(* CODESYS project retentivetimeroop_v0.0.1.1.library
   DefaultNamespace: RTimers
   Description: Standard library timers on TwinCAT count time by taking the difference between the current time from system timer and start time from system timer.
      While this is fine for most application, it is problematic for operations that require time to be retained even if the PLC is paused, stopped or turned off.
      For example, if a `TON` (Timer On-Delay) Timer is running and you stop the PLC Boot Project for a period of time, the `TON` will not resume from the point it was stopped.
      Instead it will skip time by the number of ms/secs/mins/hours it was stopped. 
      This makes it useless for applications such as tracking the length of time a PLC has been running or retaining persistent time.
      
      Retentive variants of the Standard library timers stop this from happen. They are based on PLC Task cycle time rather than system time. 
      This means they will simply stop counting when the PLC Task Cycle is stopped and will resume from where they left-off as soon as the task cycle picks up.
      All arguments behave in the same manner as those of the standard library.
   Author: Goodwill Mzumala & Victor Duran
   DocFormat: reStructuredText
   Title: Retentive Timers
   Version: 0.0.1.1
   Company: FisoThemes&Runtimevic
   Placeholder: Retentive Timers

Project tree, tasks and I/O mapping:
  libraries: Tc2_Standard, * (Beckhoff Automation GmbH); Tc2_System, * (Beckhoff Automation GmbH); Tc3_Module, * (Beckhoff Automation GmbH)
  DUTs/
    data type E_Timer_Type
    data type ST_Input
    data type ST_Output
    data type ST_PLC_TASK_INFORMATION
    data type ST_Setting
  Interfaces/
    interface I_Input: Pause, Start, StartTimer, StopTimer
    interface I_Output: Done, tElapsed
    interface I_Timer: Cyclic, Input, Output, Setting
  POUs/
    Function Block/
      Timers/
        function block FB_RStopwatch [ST]: Cyclic
        function block FB_RTimer [ST]: Cyclic
        function block FB_RTOF [ST]: Cyclic, Lerp
        function block FB_RTON [ST]: Cyclic, Lerp
        function block FB_RTP [ST]: Cyclic, Lerp
        function block FB_Stopwatch [ST]: Cyclic
        function block FB_Timer [ST]: Cyclic
      function block Timer [ST]: Cyclic, FB_exit, FB_init
      function block Timer_Abstract [ST]: Cyclic, Done, Input, Output, Pause, Setting, Start, StartTimer, StopTimer, tElapsed, tPreSet
    Functions/
      function F_Get_PLC_Task_Information [ST]
    program MAIN [ST]
  Project Information/
    function F_GetCompany [ST]
    function F_GetTitle [ST]
    function F_GetVersion [ST]
  Version/
    global variables Global_Version
*)

// DUTs/E_Timer_Type
{attribute 'qualified_only'}
{attribute 'strict'}
TYPE E_Timer_Type :
(
	RStopwatch := 0,
	RTimer,
	RTOF,
	RTON,
	RTP,
	Stopwatch,
	Timer,
	TOF,
	TON,
	TP
	
);
END_TYPE

// DUTs/ST_Input
TYPE ST_Input :
STRUCT
	bStart 		: BOOL;  // Starts timer with rising edge, resets timer with falling edge.
	bPause 		:  BOOL; // Pause Timer (TRUE), Only Pauses if IN := TRUE.
END_STRUCT
END_TYPE

// DUTs/ST_Output
TYPE ST_Output :
STRUCT
	bDone 		: BOOL; // Is TRUE, PT seconds after IN had a rising edge
	tElapsed 	: TIME; // Elapsed time
END_STRUCT
END_TYPE

// DUTs/ST_PLC_TASK_INFORMATION
TYPE ST_PLC_TASK_INFORMATION EXTENDS PlcTaskSystemInfo :
STRUCT
	tCycleTime 	: TIME; 	// Current task cycle time
	tlCycleTime : LTIME; 	// Current task cycle time in LTIME
END_STRUCT
END_TYPE

// DUTs/ST_Setting
TYPE ST_Setting :
STRUCT
	tPreSet 	: TIME; // Time to pass, before Q is set
END_STRUCT
END_TYPE

// Version/Global_Version
{attribute 'TcGenerated'}
{attribute 'no-analysis'}
{attribute 'linkalways'}
// This function has been automatically generated from the project information.
VAR_GLOBAL CONSTANT
	{attribute 'const_non_replaced'}
	stLibVersion_Retentive_Timers : ST_LibVersion := (iMajor := 0, iMinor := 0, iBuild := 1, iRevision := 1, nFlags := 0, sVersion := '0.0.1.1');
END_VAR

// Interfaces/I_Input
INTERFACE I_Input

METHOD Pause : I_Output
VAR_INPUT
	bPause 		:  BOOL; // Pause Timer (TRUE), Only Pauses if IN := TRUE.
END_VAR
END_METHOD

METHOD Start : I_Output
VAR_INPUT
	bStart 		: BOOL;  // Starts timer with rising edge, resets timer with falling edge.
END_VAR
END_METHOD

METHOD StartTimer : I_Output
VAR_INPUT
END_VAR
END_METHOD

METHOD StopTimer : I_Output
VAR_INPUT
END_VAR
END_METHOD

END_INTERFACE

// Interfaces/I_Output
INTERFACE I_Output

PROPERTY Done : BOOL
GET
END_GET
END_PROPERTY

PROPERTY tElapsed : TIME
GET
END_GET
END_PROPERTY

END_INTERFACE

// POUs/Function Block/Timer
{attribute 'hide_all_locals'}
FUNCTION_BLOCK Timer EXTENDS Timer_Abstract
VAR
	_eTimer         : E_Timer_Type;
	i_Timer			: I_Timer := 0;;
	
//	FB_RStopwatch 	: FB_RStopwatch;
//	FB_RTimer       : FB_RTimer;
//	FB_RTOF 		: FB_RTOF;
//	FB_RTON         : FB_RTON;
//	FB_RTP          : FB_RTP;
//	FB_Stopwatch 	: FB_Stopwatch;
//	FB_Timer        : FB_Timer;
	
	pRStopwatch 	: POINTER TO FB_RStopwatch;
	pRTimer       	: POINTER TO FB_RTimer;
	pRTOF 			: POINTER TO FB_RTOF;
	pRTON         	: POINTER TO FB_RTON;
	pRTP          	: POINTER TO FB_RTP;
	pStopwatch 		: POINTER TO FB_Stopwatch;
	pTimer        	: POINTER TO FB_Timer;
END_VAR

Cyclic();


METHOD Cyclic

//CASE _eTimer OF
	
//	E_Timer_Type.RStopwatch:
//		i_Timer   := FB_RStopwatch;
////	    pRStopwatch:= __NEW(FB_RStopwatch);
////		i_Timer   := pRStopwatch^;
		
////		//Release the memory
////		IF (pRStopwatch <> 0) THEN
////			__DELETE(pRStopwatch);
////			pRStopwatch := 0;
////		END_IF

//	E_Timer_Type.RTimer:
//		i_Timer   := FB_RTimer;

//	E_Timer_Type.RTOF:
//		i_Timer   := FB_RTOF;

//	E_Timer_Type.RTON:
//		i_Timer   := FB_RTON;

//	E_Timer_Type.RTP:
//		i_Timer   := FB_RTP;

//	E_Timer_Type.Stopwatch:
//		i_Timer   := FB_Stopwatch;

//	E_Timer_Type.Timer:
//		i_Timer   := FB_Timer;		
//END_CASE

IF i_Timer <> 0 THEN
	i_Timer.Input   REF= SUPER^._Input;
	i_Timer.Setting REF= SUPER^._Setting;
	i_Timer.Cyclic();
	SUPER^._Output := i_Timer.Output;
END_IF
END_METHOD

METHOD FB_exit : BOOL
VAR_INPUT
	bInCopyCode : BOOL; // if TRUE, the exit method is called for exiting an instance that is copied afterwards (online change).
END_VAR
IF (pRStopwatch <> 0) THEN
	__DELETE(pRStopwatch);
	pRStopwatch := 0;
END_IF

IF (pRTimer <> 0) THEN
	__DELETE(pRTimer);
	pRTimer := 0;
END_IF

IF (pRTOF <> 0) THEN
	__DELETE(pRTOF);
	pRTOF := 0;
END_IF

IF (pRTON <> 0) THEN
	__DELETE(pRTON);
	pRTON := 0;
END_IF

IF (pRTP <> 0) THEN
	__DELETE(pRTP);
	pRTP := 0;
END_IF

IF (pStopwatch <> 0) THEN
	__DELETE(pStopwatch);
	pStopwatch := 0;
END_IF

IF (pTimer <> 0) THEN
	__DELETE(pTimer);
	pTimer := 0;
END_IF
END_METHOD

METHOD FB_init : BOOL
VAR_INPUT
	bInitRetains : BOOL; // if TRUE, the retain variables are initialized (warm start / cold start)
	bInCopyCode : BOOL;  // if TRUE, the instance afterwards gets moved into the copy code (online change)
	eTimer      : E_Timer_Type;
END_VAR
THIS^._eTimer := eTimer;

CASE _eTimer OF
	
	E_Timer_Type.RStopwatch:
//		i_Timer   := FB_RStopwatch;
		pRStopwatch := __NEW(FB_RStopwatch);
		i_Timer := pRStopwatch^;

	E_Timer_Type.RTimer:
//		i_Timer   := FB_RTimer;
		pRTimer := __NEW(FB_RTimer);
		i_Timer := pRTimer^;

	E_Timer_Type.RTOF:
//		i_Timer   := FB_RTOF;
		pRTOF := __NEW(FB_RTOF);
		i_Timer := pRTOF^;

	E_Timer_Type.RTON:
//		i_Timer   := FB_RTON;
		pRTON := __NEW(FB_RTON);
		i_Timer := pRTON^;

	E_Timer_Type.RTP:
//		i_Timer   := FB_RTP;
		pRTP := __NEW(FB_RTP);
		i_Timer := pRTP^;

	E_Timer_Type.Stopwatch:
//		i_Timer   := FB_Stopwatch;
		pStopwatch := __NEW(FB_Stopwatch);
		i_Timer := pStopwatch^;

	E_Timer_Type.Timer:
//		i_Timer   := FB_Timer;
		pTimer := __NEW(FB_Timer);
		i_Timer := pTimer^;	
END_CASE
END_METHOD

END_FUNCTION_BLOCK

// POUs/Function Block/Timer_Abstract
{attribute 'enable_dynamic_creation'}
FUNCTION_BLOCK ABSTRACT Timer_Abstract IMPLEMENTS I_Timer, I_Input, I_Output
VAR_INPUT
END_VAR
VAR_OUTPUT
END_VAR
VAR
	_Setting 	: ST_Setting;
	_Input 		: ST_Input;
	_Output     : ST_Output;
END_VAR


METHOD ABSTRACT Cyclic
END_METHOD

PROPERTY Done : BOOL
GET
Done := _Output.bDone ;
END_GET
END_PROPERTY


PROPERTY Input : REFERENCE TO ST_Input
GET
Input REF= THIS^._Input ;
END_GET
SET
THIS^._Input := Input;
END_SET
END_PROPERTY


PROPERTY Output : REFERENCE TO ST_Output
GET
Output REF= THIS^._Output;
END_GET
END_PROPERTY

METHOD Pause : I_Output
VAR_INPUT
	bPause 		:  BOOL; // Pause Timer (TRUE), Only Pauses if IN := TRUE.
END_VAR
_Input.bPause := bPause;

Pause := THIS^;
END_METHOD


PROPERTY Setting : REFERENCE TO ST_Setting
GET
Setting REF= THIS^._Setting ;
END_GET
SET
THIS^._Setting := Setting;
END_SET
END_PROPERTY

METHOD Start : I_Output
VAR_INPUT
	bStart 		: BOOL;  // Starts timer with rising edge, resets timer with falling edge.
END_VAR
_Input.bStart := bStart;

Start := THIS^;
END_METHOD

METHOD StartTimer : I_Output
VAR_INPUT
END_VAR
_Input.bStart := TRUE;

StartTimer := THIS^;
END_METHOD

METHOD StopTimer : I_Output
VAR_INPUT
END_VAR
_Input.bStart := FALSE;

StopTimer := THIS^;
END_METHOD

PROPERTY tElapsed : TIME
GET
tElapsed := _Output.tElapsed; // Elapsed time
END_GET
END_PROPERTY

METHOD tPreSet
VAR_INPUT
	tPreSet 	: TIME; // Time to pass, before Q is set	
END_VAR
_Setting.tPreSet := tPreSet;
END_METHOD

END_FUNCTION_BLOCK

// Interfaces/I_Timer
INTERFACE I_Timer

METHOD Cyclic
END_METHOD

PROPERTY Input : REFERENCE TO ST_Input
GET
END_GET
SET
END_SET
END_PROPERTY

PROPERTY Output : REFERENCE TO ST_Output
GET
END_GET
END_PROPERTY

PROPERTY Setting : REFERENCE TO ST_Setting
GET
END_GET
SET
END_SET
END_PROPERTY

END_INTERFACE

// POUs/Function Block/Timers/FB_RStopwatch
// Retentive stopwatch
{attribute 'enable_dynamic_creation'}
FUNCTION_BLOCK INTERNAL FB_RStopwatch EXTENDS Timer_Abstract
//VAR_INPUT
//	bStart 			: BOOL;
//END_VAR
//VAR_OUTPUT
//	tElapsed 		: TIME;
//END_VAR
VAR
	stPLC_Task_Info : ST_PLC_TASK_INFORMATION;
	tAccumulator 	: TIME;
	fbTON 			: FB_RTON;
END_VAR


METHOD Cyclic
IF SUPER^._Input.bStart THEN stPLC_Task_Info := F_Get_PLC_Task_Information(); END_IF

//fbTON(tPreSet := stPLC_Task_Info.tCycleTime*2 + tAccumulator);
//fbTON(bStart := SUPER^._Input.bStart AND NOT(fbTON.output.bDone));
fbTON._Setting.tPreSet := stPLC_Task_Info.tCycleTime*2 + tAccumulator;
fbTON._Input.bStart := SUPER^._Input.bStart AND NOT(fbTON.output.bDone);
fbTON.Cyclic();

tAccumulator := fbTON.Output.tElapsed; 

IF SUPER^._Input.bStart THEN Output.tElapsed := tAccumulator; END_IF
END_METHOD

END_FUNCTION_BLOCK

// POUs/Function Block/Timers/FB_RTON
(* Retentive Timer On-Delay - implements a timer-on delay that persists if PLC cycle is stopped. 
When the input gets TRUE, elapsed time ET will run until also the output Q becomes TRUE. 
*)
{attribute 'enable_dynamic_creation'}
FUNCTION_BLOCK INTERNAL FB_RTON EXTENDS Timer_Abstract
//VAR_INPUT
//	bStart 				: BOOL; // Starts timer with rising edge, resets timer with falling edge
//	tPreSet 			: TIME; // Time to pass, before Q is set
//END_VAR
//VAR_OUTPUT
//	bDone 				: BOOL; // Is TRUE, PT seconds after IN had a rising edge
//	tElapsed 			: TIME; // Elapsed time
//END_VAR
VAR
	stPLC_Task_Info 	: ST_PLC_TASK_INFORMATION;
	tAccumulator 		: TIME;
	nLast_Cycle_Count 	: UDINT;
END_VAR


METHOD Cyclic
IF SUPER^._Input.bStart THEN
	stPLC_Task_Info := F_Get_PLC_Task_Information();
	SUPER^._Output.bDone := SUPER^._Output.tElapsed >= SUPER^._Setting.tPreSet;
	
	IF NOT(SUPER^._Output.bDone) AND ((nLast_Cycle_Count <> stPLC_Task_Info.CycleCount) OR nLast_Cycle_Count = 0) THEN
		tAccumulator := tAccumulator + stPLC_Task_Info.tCycleTime; 
		SUPER^._Output.tElapsed := LIMIT(T#0MS, THIS^.Lerp(T#0MS, SUPER^._Setting.tPreSet, TO_REAL(tAccumulator)/TO_REAL(SUPER^._Setting.tPreSet))-stPLC_Task_Info.tCycleTime, SUPER^._Setting.tPreSet);
		nLast_Cycle_Count := stPLC_Task_Info.CycleCount;
		END_IF
	RETURN;
	END_IF
tAccumulator := SUPER^._Output.tElapsed := T#0MS; SUPER^._Output.bDone := FALSE;
END_METHOD

// Linear interpolation (Lerp) - this method interpolates values between 2 time points.
METHOD PRIVATE Lerp : TIME
VAR_INPUT
	tStart 	: TIME := T#0MS; 
	tFinish : TIME;
	fPercentage : REAL; // Value must be between 0 and 1
END_VAR
// Lerp(Start, Finish, Percentage) = Start + (Finish - Start)*Percentage
Lerp := TO_TIME(TO_REAL(tStart) + TO_REAL(tFinish - tStart)*fPercentage);
END_METHOD

END_FUNCTION_BLOCK

// POUs/Functions/F_Get_PLC_Task_Information
(* Gets the infomation of the task the function is currently called on.
.. _More: https://infosys.beckhoff.com/english.php?content=../content/1033/globaldatatypes/714818699.html&id=
*)
FUNCTION F_Get_PLC_Task_Information : ST_PLC_TASK_INFORMATION
VAR_INPUT
END_VAR
VAR
	fbCurrent_Task_Index  	: GETCURTASKINDEX;
	st_TaskInfo 			: PlcTaskSystemInfo;
	stTask_Info 			: ST_PLC_TASK_INFORMATION;
END_VAR

fbCurrent_Task_Index();
st_TaskInfo 						:= TwinCAT_SystemInfoVarList._TaskInfo[fbCurrent_Task_Index.index];

stTask_Info.AdsPort 				:= st_TaskInfo.AdsPort;
stTask_Info.CycleCount 				:= st_TaskInfo.CycleCount;
stTask_Info.CycleTime 				:= st_TaskInfo.CycleTime;
stTask_Info.CycleTimeExceeded 		:= st_TaskInfo.CycleTimeExceeded;
stTask_Info.DcTaskTime 				:= st_TaskInfo.DcTaskTime;
stTask_Info.FirstCycle				:= st_TaskInfo.FirstCycle;
stTask_Info.InCallAfterOutputUpdate := st_TaskInfo.InCallAfterOutputUpdate;
stTask_Info.LastExecTime 			:= st_TaskInfo.LastExecTime;
stTask_Info.ObjId 					:= st_TaskInfo.ObjId;
stTask_Info.Priority 				:= st_TaskInfo.Priority;
stTask_Info.RTViolation 			:= st_TaskInfo.RTViolation;
stTask_Info.TaskName 				:= st_TaskInfo.TaskName;
stTask_Info.tlCycleTime 			:= TO_LTIME(st_TaskInfo.CycleTime*100);
stTask_Info.tCycleTime 				:= TO_TIME(stTask_Info.tlCycleTime);

F_Get_PLC_Task_Information 		:= stTask_Info;

END_FUNCTION

// POUs/Function Block/Timers/FB_RTimer
// Retentive Pausable Timer Function Block
{attribute 'enable_dynamic_creation'}
FUNCTION_BLOCK INTERNAL FB_RTimer EXTENDS Timer_Abstract
//VAR_INPUT
//    bStart 			: BOOL; // Start (TRUE) or Stop (FALSE) Timer 
//	bPause 			: BOOL; // Pause Timer (TRUE), Only Pauses if IN := TRUE
//    tPreSet			: TIME; // Set Time
//END_VAR
//VAR_OUTPUT
//    bDone 			: BOOL;	// Becomes TRUE after Set Time has passed
//    tElapsed 		: TIME; // Time Elapsed
//END_VAR
VAR
	fbRTON 			: FB_RTON;
END_VAR


METHOD Cyclic
IF NOT(SUPER^._Input.bStart) THEN 
	//fbRTON(bStart := FALSE, bDone => SUPER^._Output.bDone, tElapsed => SUPER^._Output.tElapsed); 
	fbRTON._Input.bStart := FALSE;
	fbRTON._Setting.tPreSet := SUPER^._Setting.tPreSet;
	fbRTON.Cyclic();
	SUPER^._Output := fbRTON.Output;
	RETURN; 
END_IF

IF SUPER^._Input.bPause THEN RETURN; END_IF;

//fbRTON(bStart := TRUE, tPreSet := SUPER^._Setting.tPreSet, bDone => SUPER^._Output.bDone, tElapsed => SUPER^._Output.tElapsed);
fbRTON._Input.bStart := TRUE;
fbRTON._Setting.tPreSet :=  SUPER^._Setting.tPreSet;
fbRTON.Cyclic();
SUPER^._Output := fbRTON.Output;
END_METHOD

END_FUNCTION_BLOCK

// POUs/Function Block/Timers/FB_RTOF
(* Retentive Timer Off-Delay - implements a timer-off delay that persists if PLC cycle is stopped. 
When the input becomes FALSE after a TRUE, the elapsed time ET will run through until the output Q becomes TRUE. 
*)
{attribute 'enable_dynamic_creation'}
FUNCTION_BLOCK INTERNAL FB_RTOF EXTENDS Timer_Abstract
//VAR_INPUT
//	bStart 				: BOOL; // Starts timer with falling edge, resets timer with rising edge
//	tPreSet 			: TIME; // Time to pass, before Q is set
//END_VAR
//VAR_OUTPUT
//	bDone 				: BOOL; // is FALSE, PT seconds after IN had a falling edge
//	tElapsed 			: TIME; // Elapsed time
//END_VAR
VAR
	stPLC_Task_Info 	: ST_PLC_TASK_INFORMATION;
	tAccumulator 		: TIME;
	nLast_Cycle_Count 	: UDINT;
	eState 				: (IDLE, RUN);
END_VAR


METHOD Cyclic
LBL_TOP: 
CASE eState OF
	IDLE: 
		IF SUPER^._Input.bStart THEN SUPER^.Output.bDone := TRUE; tAccumulator := SUPER^.Output.tElapsed := T#0MS; eState := RUN; JMP LBL_TOP; END_IF
	RUN:
		stPLC_Task_Info := F_Get_PLC_Task_Information();
		IF NOT(SUPER^._Input.bStart) AND ((nLast_Cycle_Count <> stPLC_Task_Info.CycleCount) OR nLast_Cycle_Count = 0) THEN 
			SUPER^.Output.bDone := SUPER^._Output.tElapsed <> SUPER^._Setting.tPreSet;
			IF (SUPER^._Output.tElapsed >= SUPER^._Setting.tPreSet) THEN SUPER^.Output.bDone := FALSE;  eState := IDLE; JMP LBL_TOP; END_IF
			tAccumulator := tAccumulator + stPLC_Task_Info.tCycleTime; 
			SUPER^.Output.tElapsed := LIMIT(T#0MS, THIS^.Lerp(T#0MS, SUPER^._Setting.tPreSet, TO_REAL(tAccumulator)/TO_REAL(SUPER^._Setting.tPreSet))-stPLC_Task_Info.tCycleTime, SUPER^._Setting.tPreSet);
			END_IF
		nLast_Cycle_Count := stPLC_Task_Info.CycleCount;
		IF SUPER^._Input.bStart THEN tAccumulator := SUPER^.Output.tElapsed := T#0MS;END_IF
END_CASE
END_METHOD

// Linear interpolation (Lerp) - this method interpolates values between 2 time points.
METHOD PRIVATE Lerp : TIME
VAR_INPUT
	tStart 	: TIME := T#0MS; 
	tFinish : TIME;
	fPercentage : REAL; // Value must be between 0 and 1
END_VAR
// Lerp(Start, Finish, Percentage) = Start + (Finish - Start)*Percentage
Lerp := TO_TIME(TO_REAL(tStart) + TO_REAL(tFinish - tStart)*fPercentage);
END_METHOD

END_FUNCTION_BLOCK

// POUs/Function Block/Timers/FB_RTP
(* Retentive Pulse Timer - implements a pulse time that persists if PLC cycle is stopped. 
when the input becomes TRUE, the elapsed time ET will run for the set time PT and the output Q will becomes TRUE.  
*)
{attribute 'enable_dynamic_creation'}
FUNCTION_BLOCK INTERNAL FB_RTP EXTENDS Timer_Abstract
//VAR_INPUT
//	bStart      		: BOOL; // Trigger for Start of the Signal
//    tPreSet    			: TIME; // The length of the High-Signal in ms
//END_VAR
//VAR_OUTPUT
//    bDone       		: BOOL; // The pulse
//    tElapsed      		: TIME; // The current phase of the High-Signal
//END_VAR
VAR
	stPLC_Task_Info 	: ST_PLC_TASK_INFORMATION;
	tAccumulator 		: TIME;
	nLast_Cycle_Count 	: UDINT;
	eState 				: (IDLE, RUN);
END_VAR


METHOD Cyclic
LBL_TOP:
CASE eState OF
	IDLE:
		tAccumulator := SUPER^._Output.tElapsed := T#0MS; SUPER^._Output.bDone := FALSE;
		IF SUPER^._Input.bStart THEN eState := RUN; JMP LBL_TOP; END_IF
	RUN:
		SUPER^._Output.bDone := SUPER^._Output.tElapsed < SUPER^._Setting.tPreSet;
		IF (SUPER^._Setting.tPreSet = T#0S) THEN RETURN; END_IF
		IF NOT(SUPER^._Output.bDone) AND NOT(SUPER^._Input.bStart) THEN eState := IDLE; JMP LBL_TOP; END_IF
		IF NOT(SUPER^._Output.bDone) THEN RETURN; END_IF
		stPLC_Task_Info := F_Get_PLC_Task_Information();
		IF (nLast_Cycle_Count = stPLC_Task_Info.CycleCount)THEN RETURN; END_IF
		tAccumulator := tAccumulator + stPLC_Task_Info.tCycleTime; 
		SUPER^._Output.tElapsed := LIMIT(T#0MS, THIS^.Lerp(T#0MS, SUPER^._Setting.tPreSet, TO_REAL(tAccumulator)/TO_REAL(SUPER^._Setting.tPreSet))-stPLC_Task_Info.tCycleTime, SUPER^._Setting.tPreSet);
		nLast_Cycle_Count := stPLC_Task_Info.CycleCount;	
END_CASE
END_METHOD

// Linear interpolation (Lerp) - this method interpolates values between 2 time points.
METHOD PRIVATE Lerp : TIME
VAR_INPUT
	tStart 	: TIME := T#0MS; 
	tFinish : TIME;
	fPercentage : REAL; // Value must be between 0 and 1
END_VAR
// Lerp(Start, Finish, Percentage) = Start + (Finish - Start)*Percentage
Lerp := TO_TIME(TO_REAL(tStart) + TO_REAL(tFinish - tStart)*fPercentage);
END_METHOD

END_FUNCTION_BLOCK

// POUs/Function Block/Timers/FB_Stopwatch
{attribute 'enable_dynamic_creation'}
FUNCTION_BLOCK INTERNAL FB_Stopwatch EXTENDS Timer_Abstract
//VAR_INPUT
//	bStart 			: BOOL;
//END_VAR
//VAR_OUTPUT
//	tElapsed 		: TIME;
//END_VAR
VAR
	stPLC_Task_Info : ST_PLC_TASK_INFORMATION;
	tAccumulator 	: TIME;
	fbTON 			: TON;
END_VAR


METHOD Cyclic
IF SUPER^._Input.bStart THEN stPLC_Task_Info := F_Get_PLC_Task_Information(); END_IF
fbTON(PT := stPLC_Task_Info.tCycleTime*2 + tAccumulator);
fbTON(IN := SUPER^._Input.bStart AND NOT(fbTON.Q));
tAccumulator := fbTON.ET; 
IF SUPER^._Input.bStart THEN SUPER^._Output.tElapsed := tAccumulator; END_IF
END_METHOD

END_FUNCTION_BLOCK

// POUs/Function Block/Timers/FB_Timer
// Pausable Timer Function Block
{attribute 'enable_dynamic_creation'}
FUNCTION_BLOCK INTERNAL FB_Timer EXTENDS Timer_Abstract
//VAR_INPUT
//    bStart 		: BOOL; // Start (TRUE) or Stop (FALSE) Timer 
//	bPause 		: BOOL; // Pause Timer (TRUE), Only Pauses if IN := TRUE
//    tPreSet		: TIME; // Set Time
//END_VAR
//VAR_OUTPUT
//    bDone 		: BOOL;	// Becomes TRUE after Set Time has passed
//    tElapsed 	: TIME; // Time Elapsed
//END_VAR
VAR
	fbTON 		: TON;
	tPaused 	: TIME;
	eState		: (START, PAUSE);
END_VAR


METHOD Cyclic
IF NOT(SUPER^._Input.bStart) THEN tPaused := SUPER^._Output.tElapsed := T#0MS; END_IF
fbTON(PT := SUPER^._Setting.tPreSet - tPaused, Q => SUPER^._Output.bDone);
IF SUPER^._Input.bPause THEN 
	tPaused := fbTON.ET + tPaused; 
	fbTON(IN := FALSE); 
ELSE 
	fbTON(IN := SUPER^._Input.bStart); 
	SUPER^._Output.tElapsed := fbTON.ET + tPaused; 
	END_IF
END_METHOD

END_FUNCTION_BLOCK

// POUs/MAIN
PROGRAM MAIN
VAR
	fbRStopwatch		: Timer(E_timer_type.RStopwatch);
	fbRTimer			: Timer(E_timer_type.RTimer);
	fbRTOF				: Timer(E_timer_type.RTOF);
	fbRTON				: Timer(E_timer_type.RTON);
	fbRTP				: Timer(E_timer_type.RTP);
	fbStopwatch			: Timer(E_timer_type.Stopwatch);
	fbTimer				: Timer(E_timer_type.Timer);
	
	i_Input		    : I_Input;
	counter			: INT;
	
	eStep                : (Initialization,Start_RStopwatch,RStopwatch,RTimer,RTOF,RTON,Start_RTP,RTP,Start_Stopwatch,Stopwatch,Timer);
END_VAR

// ************** Runtimevic : Víctor Durán **********************************************
// My repo GitHub OOP: https://github.com/runtimevic/OOP-IEC61131-3--Curso-Youtube
// Docu repo: https://runtimevic.github.io/OOP-IEC61131-3--Curso-Youtube/es/
// my PlayList OOP: https://www.youtube.com/playlist?list=PLEfi_hUmmSjFpfdJ6yw3B9yj7dWHYkHmQ
// email : victorduranm@hotmail.com
//*****************************************************************************************


//Settings values tPreSet Timers:
fbRTimer.Setting.tPreSet := T#3S; 	// use of Property.
fbRTOF.tPreSet(T#3S);             	// use of Method.
fbRTON.tPreSet(T#3S);             	// use of Method.
fbRTP.Setting.tPreSet := T#3S; 		// use of Property.
fbTimer.Setting.tPreSet := T#3S; 	// use of Property.
//*******************************

CASE eStep OF
	
	Initialization:
	 //fbRStopwatch.Start(bStart:=FALSE);
	  fbRStopwatch.Input.bStart := FALSE; 	// use of Property.
	  fbRTimer.Start(FALSE);             	// use of Method.
	  fbRTOF.Start(TRUE);	 				// use of Method.
	  fbRTON.Start(FALSE);	 				// use of Method.
	  fbRTP.Input.bStart := FALSE; 			// use of Property.
	  fbStopwatch.Start(FALSE);             // use of Method.
	  fbTimer.Start(FALSE);             	// use of Method.
	  counter := 0;
	  eStep:= Start_RStopwatch;
	
	Start_RStopwatch: 
		 //fbRStopwatch.Start(bStart:=TRUE); 	// use of Method.
		fbRStopwatch.Input.bStart := TRUE; 		// use of Property.
 		eStep:= RStopwatch;
	  
	RStopwatch:
	    // Example Properties.
		IF fbRStopwatch.Output.tElapsed > T#4S THEN
			fbRStopwatch.Input.bStart := FALSE;
			eStep:= RTimer;
		END_IF

	RTimer:	
	    // Example Methods.
		fbRTimer.Start(TRUE);
		IF fbRTimer.Output.bDone THEN
			fbRTimer.Start(FALSE);
			eStep:= RTOF;
		END_IF
	
	RTOF:
	   // Example Fluid Interface : https://www.plccoder.com/fluent-code/			
		IF NOT fbRTOF.Start(FALSE).Done THEN
			fbRTOF.Start(TRUE);
			eStep:= RTON;
		END_IF
		
	RTON:
		i_Input := fbRTON ; 	// use of Polymorphism.
		// Example Polymorphism with Fluid Interface.
		IF i_Input.Start(TRUE).Done THEN 
			fbRTON.Start(FALSE);
			eStep:= Start_RTP;
		END_IF	
	
	Start_RTP:
		fbRTP.Input.bStart := TRUE; 	// use of Property.
		eStep:= RTP;
		
	RTP:
		IF NOT fbRTP.Done THEN 		// use of Property.
			fbRTP.Start(FALSE);  		// use of Methods.
			eStep:= Start_Stopwatch;
		END_IF
								
	Start_Stopwatch:
		i_Input := fbRStopwatch ; 	// use of Polymorphism.
		i_Input.Start(TRUE);
		eStep:= Stopwatch;
	
	Stopwatch: 	
	   // Example Polymorphism with Fluid Interface.
	 	IF i_Input.StartTimer().tElapsed > T#3S THEN
			i_Input.StopTimer();
			eStep:= Timer;
		END_IF
		
	Timer:
		i_Input := fbTimer ; 	// use of Polymorphism.
		IF i_Input.Start(TRUE).tElapsed > T#1S AND counter < 1000 THEN
		     i_Input.Pause(TRUE);
			 counter := counter + 1;
		END_IF
		
		IF i_Input.Start(TRUE).tElapsed > T#1S AND counter >= 1000 THEN
		     i_Input.Pause(FALSE);
		END_IF
		
		IF i_Input.Start(TRUE).Done THEN //// use of Polymorphism with fluid interface...
			i_Input.Start(FALSE);
			counter := 0;
			eStep:= Initialization;
		END_IF					
END_CASE

fbRStopwatch();
fbRTimer();
fbRTOF();
fbRTON();
fbRTP();
fbStopwatch();
fbTimer();

END_PROGRAM

// Project Information/F_GetCompany
// This function has been automatically generated from the project information.
{attribute 'signature_flag' := '1073741824'}
{attribute 'TcGenerated'}
{attribute 'no-analysis'}
FUNCTION F_GetCompany : WSTRING
VAR_INPUT
	
END_VAR

F_GetCompany := "FisoThemes&Runtimevic";

END_FUNCTION

// Project Information/F_GetTitle
// This function has been automatically generated from the project information.
{attribute 'signature_flag' := '1073741824'}
{attribute 'TcGenerated'}
{attribute 'no-analysis'}
FUNCTION F_GetTitle : WSTRING
VAR_INPUT
	
END_VAR

F_GetTitle := "Retentive Timers";

END_FUNCTION

// Project Information/F_GetVersion
// This function has been automatically generated from the project information.
{attribute 'signature_flag' := '1073741824'}
{attribute 'TcGenerated'}
{attribute 'no-analysis'}
FUNCTION F_GetVersion : ST_LibVersion
VAR_INPUT
	
END_VAR

F_GetVersion.iMajor := 0;
F_GetVersion.iMinor := 0;
F_GetVersion.iBuild := 1;
F_GetVersion.iRevision := 1;
F_GetVersion.sVersion := '0.0.1.1';
F_GetVersion.nFlags := 0;

END_FUNCTION
